(* IEC 61131-3 sources: SRCI/RobotLibrary/Library/Functions/Convert/Misc, 18 files *)

(* ---- ArmConfigParameterToBytes.st ---- *)
FUNCTION ArmConfigParameterToBytes : ARRAY[0..1] of BYTE
// -------------------------------------------------------------------------
//  SRCI Robot Library
// -------------------------------------------------------------------------
//
//  Object:      ArmConfigParameterToBytes
//  Author:      Thorsten Brach
//  Date:        2025-01-30
//
//  Description:
//
//
//  Copyright:
//    (C) 2025 Thorsten Brach. All rights reserved
//             Licensed under the LGPL-3.0 license.
//
//  Disclaimer:
//    This project is provided without any guarantee and can be used for
//    private and commercial purposes. Any use is at the user’s
//    own risk and responsibility.
//
// -------------------------------------------------------------------------
VAR_INPUT
 /// ArmConfigParameter
 Value: ArmConfigParameter;
END_VAR

  ArmConfigParameterToBytes[0].0 := Value.Shoulder.0;
  ArmConfigParameterToBytes[0].1 := Value.Shoulder.1;
  ArmConfigParameterToBytes[0].2 := Value.Shoulder.2;
  ArmConfigParameterToBytes[0].3 := Value.Shoulder.3;
  ArmConfigParameterToBytes[0].4 := Value.Elbow.0;
  ArmConfigParameterToBytes[0].5 := Value.Elbow.1;
  ArmConfigParameterToBytes[0].6 := Value.Elbow.2;
  ArmConfigParameterToBytes[0].7 := Value.Elbow.3;
  ArmConfigParameterToBytes[1].0 := Value.Wrist.0;
  ArmConfigParameterToBytes[1].1 := Value.Wrist.1;
  ArmConfigParameterToBytes[1].2 := Value.Wrist.2;
  ArmConfigParameterToBytes[1].3 := Value.Wrist.3;
  ArmConfigParameterToBytes[1].4 := FALSE;
  ArmConfigParameterToBytes[1].5 := FALSE;
  ArmConfigParameterToBytes[1].6 := FALSE;
  ArmConfigParameterToBytes[1].7 := FALSE;

END_FUNCTION

(* ---- BytesToRCSupportedFunctions.st ---- *)
FUNCTION BytesToRCSupportedFunctions : RCSupportedFunctions
// -------------------------------------------------------------------------
//  SRCI Robot Library
// -------------------------------------------------------------------------
//
//  Object:      BytesToRCSupportedFunctions
//  Author:      Thorsten Brach
//  Date:        2024-12-18
//
//  Description:
//
//
//  Copyright:
//    (C) 2024 Thorsten Brach. All rights reserved
//             Licensed under the LGPL-3.0 license.
//
//  Disclaimer:
//    This project is provided without any guarantee and can be used for
//    private and commercial purposes. Any use is at the user’s
//    own risk and responsibility.
//
// -------------------------------------------------------------------------
VAR_INPUT
  Bytes : ARRAY [0..18] OF BYTE;
END_VAR

  // Byte 00 - Bit 0
  BytesToRCSupportedFunctions.Reserved                   := Bytes[00].0;
  // Byte 00 - Bit 1
  BytesToRCSupportedFunctions.ReadRobotData              := Bytes[00].1;
  // Byte 00 - Bit 2
  BytesToRCSupportedFunctions.EnableRobot                := Bytes[00].2;
  // Byte 00 - Bit 3
  BytesToRCSupportedFunctions.GroupReset                 := Bytes[00].3;
  // Byte 00 - Bit 4
  BytesToRCSupportedFunctions.ReadActualPosition         := Bytes[00].4;
  // Byte 00 - Bit 5
  BytesToRCSupportedFunctions.ReadActualPositionCyclic   := Bytes[00].5;
  // Byte 00 - Bit 6
  BytesToRCSupportedFunctions.ExchangeConfiguration      := Bytes[00].6;
  // Byte 00 - Bit 7
  BytesToRCSupportedFunctions.SetSequence                := Bytes[00].7;

  // Byte 01 - Bit 0
  BytesToRCSupportedFunctions.ChangeSpeedOverride        := Bytes[01].0;
  // Byte 01 - Bit 1
  BytesToRCSupportedFunctions.ReadMessages               := Bytes[01].1;
  // Byte 01 - Bit 2
  BytesToRCSupportedFunctions.ReadRobotReferenceDynamics := Bytes[01].2;
  // Byte 01 - Bit 3
  BytesToRCSupportedFunctions.WriteFrameData             := Bytes[01].3;
  // Byte 01 - Bit 4
  BytesToRCSupportedFunctions.WriteToolData              := Bytes[01].4;
  // Byte 01 - Bit 5
  BytesToRCSupportedFunctions.WriteLoadData              := Bytes[01].5;
  // Byte 01 - Bit 6
  BytesToRCSupportedFunctions.WriteRobotReferenceDynamics:= Bytes[01].6;
  // Byte 01 - Bit 7
  BytesToRCSupportedFunctions.WriteRobotDefaultDynamics  := Bytes[01].7;

  // Byte 02 - Bit 0
  BytesToRCSupportedFunctions.ReadRobotDefaultDynamics   := Bytes[02].0;
  // Byte 02 - Bit 1
  BytesToRCSupportedFunctions.ReadFrameData              := Bytes[02].1;
  // Byte 02 - Bit 2
  BytesToRCSupportedFunctions.ReadToolData               := Bytes[02].2;
  // Byte 02 - Bit 3
  BytesToRCSupportedFunctions.ReadLoadData               := Bytes[02].3;
  // Byte 02 - Bit 4
  BytesToRCSupportedFunctions.ReadRobotSWLimits          := Bytes[02].4;
  // Byte 02 - Bit 5
  BytesToRCSupportedFunctions.GroupJog                   := Bytes[02].5;
  // Byte 02 - Bit 6
  BytesToRCSupportedFunctions.MoveLinearAbsolute         := Bytes[02].6;
  // Byte 02 - Bit 7
  BytesToRCSupportedFunctions.MoveDirectAbsolute         := Bytes[02].7;

  // Byte 03 - Bit 0
  BytesToRCSupportedFunctions.MoveAxesAbsolute           := Bytes[03].0;
  // Byte 03 - Bit 1
  BytesToRCSupportedFunctions.GroupStop                  := Bytes[03].1;
  // Byte 03 - Bit 2
  BytesToRCSupportedFunctions.GroupContinue              := Bytes[03].2;
  // Byte 03 - Bit 3
  BytesToRCSupportedFunctions.GroupInterrupt             := Bytes[03].3;
  // Byte 03 - Bit 4
  BytesToRCSupportedFunctions.ReturnToPrimary            := Bytes[03].4;
  // Byte 03 - Bit 5
  BytesToRCSupportedFunctions.MoveLinearAbsoluteJ        := Bytes[03].5;
  // Byte 03 - Bit 6
  BytesToRCSupportedFunctions.MoveDirectRelative         := Bytes[03].6;
  // Byte 03 - Bit 7
  BytesToRCSupportedFunctions.MoveAxesRelative           := Bytes[03].7;

  // Byte 04 - Bit 0
  BytesToRCSupportedFunctions.MoveCircularAbsolute       := Bytes[04].0;
  // Byte 04 - Bit 1
  BytesToRCSupportedFunctions.MoveCircularRelative       := Bytes[04].1;
  // Byte 04 - Bit 2
  BytesToRCSupportedFunctions.MoveLinearOffset           := Bytes[04].2;
  // Byte 04 - Bit 3
  BytesToRCSupportedFunctions.MoveDirectOffset           := Bytes[04].3;
  // Byte 04 - Bit 4
  BytesToRCSupportedFunctions.WaitTime                   := Bytes[04].4;
  // Byte 04 - Bit 5
  BytesToRCSupportedFunctions.ReadDigitalInputs          := Bytes[04].5;
  // Byte 04 - Bit 6
  BytesToRCSupportedFunctions.ReadDigitalOutputs         := Bytes[04].6;
  // Byte 04 - Bit 7
  BytesToRCSupportedFunctions.WriteDigitalOutputs        := Bytes[04].7;

  // Byte 05 - Bit 0
  BytesToRCSupportedFunctions.ReadIntegers               := Bytes[05].0;
  // Byte 05 - Bit 1
  BytesToRCSupportedFunctions.ReadReals                  := Bytes[05].1;
  // Byte 05 - Bit 2
  BytesToRCSupportedFunctions.WriteIntegers              := Bytes[05].2;
  // Byte 05 - Bit 3
  BytesToRCSupportedFunctions.WriteReals                 := Bytes[05].3;
  // Byte 05 - Bit 4
  BytesToRCSupportedFunctions.MoveLinearCam              := Bytes[05].4;
  // Byte 05 - Bit 5
  BytesToRCSupportedFunctions.MoveDirectCam              := Bytes[05].5;
  // Byte 05 - Bit 6
  BytesToRCSupportedFunctions.MoveCircularCam            := Bytes[05].6;
  // Byte 05 - Bit 7
  BytesToRCSupportedFunctions.SetTriggerRegister         := Bytes[05].7;

  // Byte 06 - Bit 0
  BytesToRCSupportedFunctions.SetTriggerLimit            := Bytes[06].0;
  // Byte 06 - Bit 1
  BytesToRCSupportedFunctions.SetTriggerUser             := Bytes[06].1;
  // Byte 06 - Bit 2
  BytesToRCSupportedFunctions.SetTriggerError            := Bytes[06].2;
  // Byte 06 - Bit 3
  BytesToRCSupportedFunctions.ReactAtTrigger             := Bytes[06].3;
  // Byte 06 - Bit 4
  BytesToRCSupportedFunctions.WaitForTrigger             := Bytes[06].4;
  // Byte 06 - Bit 5
  BytesToRCSupportedFunctions.ReadSystemVariable         := Bytes[06].5;
  // Byte 06 - Bit 6
  BytesToRCSupportedFunctions.WriteSystemVariable        := Bytes[06].6;
  // Byte 06 - Bit 7
  BytesToRCSupportedFunctions.CalculateForwardKinematic  := Bytes[06].7;

  // Byte 07 - Bit 0
  BytesToRCSupportedFunctions.CalculateInverseKinematic  := Bytes[07].0;
  // Byte 07 - Bit 1
  BytesToRCSupportedFunctions.CalculateCartesianPosition := Bytes[07].1;
  // Byte 07 - Bit 2
  BytesToRCSupportedFunctions.CalculateTool              := Bytes[07].2;
  // Byte 07 - Bit 3
  BytesToRCSupportedFunctions.CalculateFrame             := Bytes[07].3;
  // Byte 07 - Bit 4
  BytesToRCSupportedFunctions.ActivateNextCommand        := Bytes[07].4;
  // Byte 07 - Bit 5
  BytesToRCSupportedFunctions.ShiftPosition              := Bytes[07].5;
  // Byte 07 - Bit 6
  BytesToRCSupportedFunctions.CallSubprogram             := Bytes[07].6;
  // Byte 07 - Bit 7
  BytesToRCSupportedFunctions.MoveLinearRelative         := Bytes[07].7;

  // Byte 08 - Bit 0
  BytesToRCSupportedFunctions.WriteCallSubprogramCyclic  := Bytes[08].0;
  // Byte 08 - Bit 1
  BytesToRCSupportedFunctions.ReadCallSubprogramCyclic   := Bytes[08].1;
  // Byte 08 - Bit 2
  BytesToRCSupportedFunctions.StopSubprogram             := Bytes[08].2;
  // Byte 08 - Bit 3
  BytesToRCSupportedFunctions.ReadDHParameter            := Bytes[08].3;
  // Byte 08 - Bit 4
  BytesToRCSupportedFunctions.RestartController          := Bytes[08].4;
  // Byte 08 - Bit 5
  BytesToRCSupportedFunctions.ReadActualTCPVelocity      := Bytes[08].5;
  // Byte 08 - Bit 6
  BytesToRCSupportedFunctions.UserLogin                  := Bytes[08].6;
  // Byte 08 - Bit 7
  BytesToRCSupportedFunctions.SwitchLanguage             := Bytes[08].7;

  // Byte 09 - Bit 0
  BytesToRCSupportedFunctions.WriteRobotSWLimits         := Bytes[09].0;
  // Byte 09 - Bit 1
  BytesToRCSupportedFunctions.SetOperationMode           := Bytes[09].1;
  // Byte 09 - Bit 2
  BytesToRCSupportedFunctions.ReadWorkArea               := Bytes[09].2;
  // Byte 09 - Bit 3
  BytesToRCSupportedFunctions.WriteWorkArea              := Bytes[09].3;
  // Byte 09 - Bit 4
  BytesToRCSupportedFunctions.ActivateWorkArea           := Bytes[09].4;
  // Byte 09 - Bit 5
  BytesToRCSupportedFunctions.MonitorWorkArea            := Bytes[09].5;
  // Byte 09 - Bit 6
  BytesToRCSupportedFunctions.MoveApproachLinear         := Bytes[09].6;
  // Byte 09 - Bit 7
  BytesToRCSupportedFunctions.MoveDepartLinear           := Bytes[09].7;

  // Byte 10 - Bit 0
  BytesToRCSupportedFunctions.MoveApproachDirect         := Bytes[10].0;
  // Byte 10 - Bit 1
  BytesToRCSupportedFunctions.MoveDepartDirect           := Bytes[10].1;
  // Byte 10 - Bit 2
  BytesToRCSupportedFunctions.SearchHardstop             := Bytes[10].2;
  // Byte 10 - Bit 3
  BytesToRCSupportedFunctions.SearchHardstopJ            := Bytes[10].3;
  // Byte 10 - Bit 4
  BytesToRCSupportedFunctions.MovePickPlaceLinear        := Bytes[10].4;
  // Byte 10 - Bit 5
  BytesToRCSupportedFunctions.MovePickPlaceDirect        := Bytes[10].5;
  // Byte 10 - Bit 6
  BytesToRCSupportedFunctions.ActivateConveyorTracking   := Bytes[10].6;
  // Byte 10 - Bit 7
  BytesToRCSupportedFunctions.RedefineTrackingPosition   := Bytes[10].7;

  // Byte 11 - Bit 0
  BytesToRCSupportedFunctions.SyncToConveyor             := Bytes[11].0;
  // Byte 11 - Bit 1
  BytesToRCSupportedFunctions.ConfigureConveyor          := Bytes[11].1;
  // Byte 11 - Bit 2
  BytesToRCSupportedFunctions.MoveSuperImposed           := Bytes[11].2;
  // Byte 11 - Bit 3
  BytesToRCSupportedFunctions.MoveSuperImposedDynamic    := Bytes[11].3;
  // Byte 11 - Bit 4
  BytesToRCSupportedFunctions.ReadAnalogInput            := Bytes[11].4;
  // Byte 11 - Bit 5
  BytesToRCSupportedFunctions.ReadAnalogOutput           := Bytes[11].5;
  // Byte 11 - Bit 6
  BytesToRCSupportedFunctions.WriteAnalogOutput          := Bytes[11].6;
  // Byte 11 - Bit 7
  BytesToRCSupportedFunctions.MeasuringInput             := Bytes[11].7;

  // Byte 12 - Bit 0
  BytesToRCSupportedFunctions.AbortMeasuringInput        := Bytes[12].0;
  // Byte 12 - Bit 1
  BytesToRCSupportedFunctions.SetTriggerMotion           := Bytes[12].1;
  // Byte 12 - Bit 2
  BytesToRCSupportedFunctions.OpenBrake                  := Bytes[12].2;
  // Byte 12 - Bit 3
  BytesToRCSupportedFunctions.PathAccuracyMode           := Bytes[12].3;
  // Byte 12 - Bit 4
  BytesToRCSupportedFunctions.AvoidSingularity           := Bytes[12].4;
  // Byte 12 - Bit 5
  BytesToRCSupportedFunctions.ForceControl               := Bytes[12].5;
  // Byte 12 - Bit 6
  BytesToRCSupportedFunctions.ForceLimit                 := Bytes[12].6;
  // Byte 12 - Bit 7
  BytesToRCSupportedFunctions.ReadActualForce            := Bytes[12].7;

  // Byte 13 - Bit 0
  BytesToRCSupportedFunctions.BrakeTest                  := Bytes[13].0;
  // Byte 13 - Bit 1
  BytesToRCSupportedFunctions.SoftSwitchTCP              := Bytes[13].1;
  // Byte 13 - Bit 2
  BytesToRCSupportedFunctions.CreateSpline               := Bytes[13].2;
  // Byte 13 - Bit 3
  BytesToRCSupportedFunctions.DeleteSpline               := Bytes[13].3;
  // Byte 13 - Bit 4
  BytesToRCSupportedFunctions.MoveSpline                 := Bytes[13].4;
  // Byte 13 - Bit 5
  BytesToRCSupportedFunctions.DynamicSpline              := Bytes[13].5;
  // Byte 13 - Bit 6
  BytesToRCSupportedFunctions.LoadMeasurementAutomatic   := Bytes[13].6;
  // Byte 13 - Bit 7
  BytesToRCSupportedFunctions.LoadMeasurementSequential  := Bytes[13].7;

  // Byte 14 - Bit 0
  BytesToRCSupportedFunctions.CollisionDetection         := Bytes[14].0;
  // Byte 14 - Bit 1
  BytesToRCSupportedFunctions.FreeDrive                  := Bytes[14].1;
  // Byte 14 - Bit 2
  BytesToRCSupportedFunctions.UnitMeasurement            := Bytes[14].2;
  // Byte 14 - Bit 3
  BytesToRCSupportedFunctions.Byte14Bit03                := Bytes[14].3;
  // Byte 14 - Bit 4
  BytesToRCSupportedFunctions.Byte14Bit04                := Bytes[14].4;
  // Byte 14 - Bit 5
  BytesToRCSupportedFunctions.Byte14Bit05                := Bytes[14].5;
  // Byte 14 - Bit 6
  BytesToRCSupportedFunctions.Byte14Bit06                := Bytes[14].6;
  // Byte 14 - Bit 7
  BytesToRCSupportedFunctions.Byte14Bit07                := Bytes[14].7;

  // Byte 15 - Bit 0
  BytesToRCSupportedFunctions.Byte15Bit00                := Bytes[15].0;
  // Byte 15 - Bit 1
  BytesToRCSupportedFunctions.Byte15Bit01                := Bytes[15].1;
  // Byte 15 - Bit 2
  BytesToRCSupportedFunctions.Byte15Bit02                := Bytes[15].2;
  // Byte 15 - Bit 3
  BytesToRCSupportedFunctions.Byte15Bit03                := Bytes[15].3;
  // Byte 15 - Bit 4
  BytesToRCSupportedFunctions.Byte15Bit04                := Bytes[15].4;
  // Byte 15 - Bit 5
  BytesToRCSupportedFunctions.Byte15Bit05                := Bytes[15].5;
  // Byte 15 - Bit 6
  BytesToRCSupportedFunctions.Byte15Bit06                := Bytes[15].6;
  // Byte 15 - Bit 7
  BytesToRCSupportedFunctions.Byte15Bit07                := Bytes[15].7;

  // Byte 16 - Bit 0
  BytesToRCSupportedFunctions.Byte16Bit00                := Bytes[16].0;
  // Byte 15 - Bit 1
  BytesToRCSupportedFunctions.Byte16Bit01                := Bytes[16].1;
  // Byte 15 - Bit 2
  BytesToRCSupportedFunctions.Byte16Bit02                := Bytes[16].2;
  // Byte 15 - Bit 3
  BytesToRCSupportedFunctions.Byte16Bit03                := Bytes[16].3;
  // Byte 15 - Bit 4
  BytesToRCSupportedFunctions.Byte16Bit04                := Bytes[16].4;
  // Byte 15 - Bit 5
  BytesToRCSupportedFunctions.Byte16Bit05                := Bytes[16].5;
  // Byte 15 - Bit 6
  BytesToRCSupportedFunctions.Byte16Bit06                := Bytes[16].6;
  // Byte 15 - Bit 7
  BytesToRCSupportedFunctions.Byte16Bit07                := Bytes[16].7;

  // Byte 17 - Bit 0
  BytesToRCSupportedFunctions.Byte17Bit00                := Bytes[17].0;
  // Byte 17 - Bit 1
  BytesToRCSupportedFunctions.Byte17Bit01                := Bytes[17].1;
  // Byte 17 - Bit 2
  BytesToRCSupportedFunctions.Byte17Bit02                := Bytes[17].2;
  // Byte 17 - Bit 3
  BytesToRCSupportedFunctions.Byte17Bit03                := Bytes[17].3;
  // Byte 17 - Bit 4
  BytesToRCSupportedFunctions.Byte17Bit04                := Bytes[17].4;
  // Byte 17 - Bit 5
  BytesToRCSupportedFunctions.Byte17Bit05                := Bytes[17].5;
  // Byte 17 - Bit 6
  BytesToRCSupportedFunctions.Byte17Bit06                := Bytes[17].6;
  // Byte 17 - Bit 7
  BytesToRCSupportedFunctions.Byte17Bit07                := Bytes[17].7;

  // Byte 18 - Bit 0
  BytesToRCSupportedFunctions.Byte18Bit00                := Bytes[18].0;
  // Byte 18 - Bit 1
  BytesToRCSupportedFunctions.Byte18Bit01                := Bytes[18].1;
  // Byte 18 - Bit 2
  BytesToRCSupportedFunctions.Byte18Bit02                := Bytes[18].2;
  // Byte 18 - Bit 3
  BytesToRCSupportedFunctions.Byte18Bit03                := Bytes[18].3;
  // Byte 18 - Bit 4
  BytesToRCSupportedFunctions.Byte18Bit04                := Bytes[18].4;
  // Byte 18 - Bit 5
  BytesToRCSupportedFunctions.Byte18Bit05                := Bytes[18].5;
  // Byte 18 - Bit 6
  BytesToRCSupportedFunctions.Byte18Bit06                := Bytes[18].6;
  // Byte 18 - Bit 7
  BytesToRCSupportedFunctions.Byte18Bit07                := Bytes[18].7;

END_FUNCTION

(* ---- ByteToAxisExternalUnit.st ---- *)
FUNCTION ByteToAxisExternalUnit : AxisExternalUnit
// -------------------------------------------------------------------------
//  SRCI Robot Library
// -------------------------------------------------------------------------
//
//  Object:      ByteToAxisExternalUnit
//  Author:      Thorsten Brach
//  Date:        2025-03-23
//
//  Description:
//
//
//  Copyright:
//    (C) 2025 Thorsten Brach. All rights reserved
//             Licensed under the LGPL-3.0 license.
//
//  Disclaimer:
//    This project is provided without any guarantee and can be used for
//    private and commercial purposes. Any use is at the user’s
//    own risk and responsibility.
//
// -------------------------------------------------------------------------
VAR_INPUT
  AxisExternalUnit : BYTE;
END_VAR

  ByteToAxisExternalUnit.E1.0 := AxisExternalUnit.1;
  ByteToAxisExternalUnit.E2.0 := AxisExternalUnit.2;
  ByteToAxisExternalUnit.E3.0 := AxisExternalUnit.3;
  ByteToAxisExternalUnit.E4.0 := AxisExternalUnit.4;
  ByteToAxisExternalUnit.E5.0 := AxisExternalUnit.5;
  ByteToAxisExternalUnit.E6.0 := AxisExternalUnit.6;

END_FUNCTION

(* ---- ByteToAxisExternalUsed.st ---- *)
FUNCTION ByteToAxisExternalUsed : AxisExternalUsed
// -------------------------------------------------------------------------
//  SRCI Robot Library
// -------------------------------------------------------------------------
//
//  Object:      ByteToAxisExternalUsed
//  Author:      Thorsten Brach
//  Date:        2025-03-23
//
//  Description:
//
//
//  Copyright:
//    (C) 2025 Thorsten Brach. All rights reserved
//             Licensed under the LGPL-3.0 license.
//
//  Disclaimer:
//    This project is provided without any guarantee and can be used for
//    private and commercial purposes. Any use is at the user’s
//    own risk and responsibility.
//
// -------------------------------------------------------------------------
VAR_INPUT
  AxisExternalUsed : BYTE;
END_VAR

  ByteToAxisExternalUsed.E1 := AxisExternalUsed.1;
  ByteToAxisExternalUsed.E2 := AxisExternalUsed.2;
  ByteToAxisExternalUsed.E3 := AxisExternalUsed.3;
  ByteToAxisExternalUsed.E4 := AxisExternalUsed.4;
  ByteToAxisExternalUsed.E5 := AxisExternalUsed.5;
  ByteToAxisExternalUsed.E6 := AxisExternalUsed.6;

END_FUNCTION

(* ---- ByteToAxisJointUnit.st ---- *)
FUNCTION ByteToAxisJointUnit : AxisJointUnit
// -------------------------------------------------------------------------
//  SRCI Robot Library
// -------------------------------------------------------------------------
//
//  Object:      ByteToAxisJointUnit
//  Author:      Thorsten Brach
//  Date:        2025-03-23
//
//  Description:
//
//
//  Copyright:
//    (C) 2025 Thorsten Brach. All rights reserved
//             Licensed under the LGPL-3.0 license.
//
//  Disclaimer:
//    This project is provided without any guarantee and can be used for
//    private and commercial purposes. Any use is at the user’s
//    own risk and responsibility.
//
// -------------------------------------------------------------------------
VAR_INPUT
  AxisJointUnit : BYTE;
END_VAR

  ByteToAxisJointUnit.J2.0 := AxisJointUnit.1;
  ByteToAxisJointUnit.J2.0 := AxisJointUnit.2;
  ByteToAxisJointUnit.J3.0 := AxisJointUnit.3;
  ByteToAxisJointUnit.J4.0 := AxisJointUnit.4;
  ByteToAxisJointUnit.J5.0 := AxisJointUnit.5;
  ByteToAxisJointUnit.J6.0 := AxisJointUnit.6;

END_FUNCTION

(* ---- ByteToAxisJointUsed.st ---- *)
FUNCTION ByteToAxisJointUsed : AxisJointUsed
// -------------------------------------------------------------------------
//  SRCI Robot Library
// -------------------------------------------------------------------------
//
//  Object:      ByteToAxisJointUsed
//  Author:      Thorsten Brach
//  Date:        2025-03-23
//
//  Description:
//
//
//  Copyright:
//    (C) 2025 Thorsten Brach. All rights reserved
//             Licensed under the LGPL-3.0 license.
//
//  Disclaimer:
//    This project is provided without any guarantee and can be used for
//    private and commercial purposes. Any use is at the user’s
//    own risk and responsibility.
//
// -------------------------------------------------------------------------
VAR_INPUT
  AxisJointUsed : BYTE;
END_VAR

  ByteToAxisJointUsed.J1 := AxisJointUsed.1;
  ByteToAxisJointUsed.J2 := AxisJointUsed.2;
  ByteToAxisJointUsed.J3 := AxisJointUsed.3;
  ByteToAxisJointUsed.J4 := AxisJointUsed.4;
  ByteToAxisJointUsed.J5 := AxisJointUsed.5;
  ByteToAxisJointUsed.J6 := AxisJointUsed.6;

END_FUNCTION

(* ---- CombineBytesToUint.st ---- *)
FUNCTION CombineBytesToUint : UINT
// -------------------------------------------------------------------------
//  SRCI Robot Library
// -------------------------------------------------------------------------
//
//  Object:      CombineBytes
//  Author:      Thorsten Brach
//  Date:        2024-09-03
//
//  Description:
//
//
//  Copyright:
//    (C) 2024 Thorsten Brach. All rights reserved
//             Licensed under the LGPL-3.0 license.
//
//  Disclaimer:
//    This project is provided without any guarantee and can be used for
//    private and commercial purposes. Any use is at the user’s
//    own risk and responsibility.
//
// -------------------------------------------------------------------------
VAR_INPUT
  /// Byte to add as high byte
  HiByte : BYTE;
  /// Byte to add as low byte
  LoByte : BYTE;
END_VAR

  CombineBytesToUint.0  := LoByte.0;
  CombineBytesToUint.1  := LoByte.1;
  CombineBytesToUint.2  := LoByte.2;
  CombineBytesToUint.3  := LoByte.3;
  CombineBytesToUint.4  := LoByte.4;
  CombineBytesToUint.5  := LoByte.5;
  CombineBytesToUint.6  := LoByte.6;
  CombineBytesToUint.7  := LoByte.7;

  CombineBytesToUint.8  := HiByte.0;
  CombineBytesToUint.9  := HiByte.1;
  CombineBytesToUint.10 := HiByte.2;
  CombineBytesToUint.11 := HiByte.3;
  CombineBytesToUint.12 := HiByte.4;
  CombineBytesToUint.13 := HiByte.5;
  CombineBytesToUint.14 := HiByte.6;
  CombineBytesToUint.15 := HiByte.7;

END_FUNCTION

(* ---- CombineHalfSints.st ---- *)
FUNCTION CombineHalfSints : USINT
// -------------------------------------------------------------------------
//  SRCI Robot Library
// -------------------------------------------------------------------------
//
//  Object:      CombineHalfSints
//  Author:      Thorsten Brach
//  Date:        2025-02-02
//
//  Description:
//
//
//  Copyright:
//    (C) 2025 Thorsten Brach. All rights reserved
//             Licensed under the LGPL-3.0 license.
//
//  Disclaimer:
//    This project is provided without any guarantee and can be used for
//    private and commercial purposes. Any use is at the user’s
//    own risk and responsibility.
//
// -------------------------------------------------------------------------
VAR_INPUT
  /// Half-Sint to add to the upper 4 Bit
  HalfSintHi : SINT;
  /// Half-Sint to add to the lower 4 Bit
  HalfSintLo : SINT;
END_VAR

  // merage ParSeq and Priority to combined variable
  CombineHalfSints.0 := HalfSintLo.0;
  CombineHalfSints.1 := HalfSintLo.1;
  CombineHalfSints.2 := HalfSintLo.2;
  CombineHalfSints.3 := HalfSintLo.3;

  CombineHalfSints.4 := HalfSintHi.0;
  CombineHalfSints.5 := HalfSintHi.1;
  CombineHalfSints.6 := HalfSintHi.2;
  CombineHalfSints.7 := HalfSintHi.3;

END_FUNCTION

(* ---- DwordToRaStatusWord.st ---- *)
FUNCTION DwordToRaStatusWord : RaStatusWord
// -------------------------------------------------------------------------
//  SRCI Robot Library
// -------------------------------------------------------------------------
//
//  Object:      DwordToRaStatusWord
//  Author:      Thorsten Brach
//  Date:        2024-11-16
//
//  Description:
//
//
//  Copyright:
//    (C) 2024 Thorsten Brach. All rights reserved
//             Licensed under the LGPL-3.0 license.
//
//  Disclaimer:
//    This project is provided without any guarantee and can be used for
//    private and commercial purposes. Any use is at the user’s
//    own risk and responsibility.
//
// -------------------------------------------------------------------------
VAR_INPUT
  /// Value
  Value : DWORD;
END_VAR

  DwordToRaStatusWord.IsMoving                 := Value.00;
  DwordToRaStatusWord.PrimarySequencePaused    := Value.01;
  DwordToRaStatusWord.InPrimaryPos             := Value.02;
  DwordToRaStatusWord.SecondarySequenceActive  := Value.03;
  DwordToRaStatusWord.IsBlending               := Value.04;
  DwordToRaStatusWord.ErrorPending             := Value.05;
  DwordToRaStatusWord.RestartInProgress        := Value.06;
  DwordToRaStatusWord.Enabled                  := Value.07;
  DwordToRaStatusWord.RaSequenceState.0        := Value.08;
  DwordToRaStatusWord.RaSequenceState.1        := Value.09;
  DwordToRaStatusWord.OperationMode.0          := Value.10;
  DwordToRaStatusWord.OperationMode.1          := Value.11;
  DwordToRaStatusWord.OperationMode.2          := Value.12;
  DwordToRaStatusWord.CollisionDetectedEnabled := Value.13;
  DwordToRaStatusWord.CollisionDetected        := Value.14;
  DwordToRaStatusWord.RestartRequested         := Value.15;
  DwordToRaStatusWord.Accelerating             := Value.16;
  DwordToRaStatusWord.Decelerating             := Value.17;
  DwordToRaStatusWord.ConstantVelocity         := Value.18;
  DwordToRaStatusWord.Bit19                    := Value.19;
  DwordToRaStatusWord.Bit20                    := Value.20;
  DwordToRaStatusWord.Bit21                    := Value.21;
  DwordToRaStatusWord.Bit22                    := Value.22;
  DwordToRaStatusWord.Bit23                    := Value.23;
  DwordToRaStatusWord.Bit24                    := Value.24;
  DwordToRaStatusWord.Bit25                    := Value.25;
  DwordToRaStatusWord.Bit26                    := Value.26;
  DwordToRaStatusWord.Bit27                    := Value.27;
  DwordToRaStatusWord.Bit28                    := Value.28;
  DwordToRaStatusWord.Bit29                    := Value.29;
  DwordToRaStatusWord.Bit30                    := Value.30;
  DwordToRaStatusWord.Bit31                    := Value.31;

END_FUNCTION

(* ---- PERCENT_INT_TO_REAL.st ---- *)
FUNCTION PERCENT_INT_TO_REAL : REAL
// -------------------------------------------------------------------------
//  SRCI Robot Library
// -------------------------------------------------------------------------
//
//  Object:      PERCENT_INT_TO_REAL
//  Author:      Thorsten Brach
//  Date:        2025-02-07
//
//  Description:
//
//
//  Copyright:
//    (C) 2025 Thorsten Brach. All rights reserved
//             Licensed under the LGPL-3.0 license.
//
//  Disclaimer:
//    This project is provided without any guarantee and can be used for
//    private and commercial purposes. Any use is at the user’s
//    own risk and responsibility.
//
// -------------------------------------------------------------------------
VAR_INPUT
  /// Percent value to convert
  Value    : INT;
  /// value is an optional parameter ?
  IsOptional : BOOL;
END_VAR

  IF ( Value = 16#FFFF ) AND (IsOptional)// 16#FFFF for not supported values
  THEN
    PERCENT_INT_TO_REAL := -1.0;
    RETURN;
  END_IF

  PERCENT_INT_TO_REAL := INT_TO_REAL(Value) / RobotLibraryConstants.REAL_CONVERSION_FACTOR; {warning 'ToDo: check conversation is correct ?'}

END_FUNCTION

(* ---- PERCENT_UINT_TO_REAL.st ---- *)
FUNCTION PERCENT_UINT_TO_REAL : REAL
// -------------------------------------------------------------------------
//  SRCI Robot Library
// -------------------------------------------------------------------------
//
//  Object:      PERCENT_UINT_TO_REAL
//  Author:      Thorsten Brach
//  Date:        2025-04-02
//
//  Description:
//
//
//  Copyright:
//    (C) 2025 Thorsten Brach. All rights reserved
//             Licensed under the LGPL-3.0 license.
//
//  Disclaimer:
//    This project is provided without any guarantee and can be used for
//    private and commercial purposes. Any use is at the user’s
//    own risk and responsibility.
//
// -------------------------------------------------------------------------
VAR_INPUT
  /// Percent value to convert
  Value    : UINT;
  /// value is an optional parameter ?
  IsOptional : BOOL;
END_VAR

  IF (( Value = 16#FFFF_FFFF ) AND (IsOptional)) OR // 16#FFFF_FFFF for not supported values
     (( Value = 16#0000_FFFF ) AND (IsOptional))    // 16#0000_FFFF for not supported values
  THEN
    PERCENT_UINT_TO_REAL := -1.0;
    RETURN;
  END_IF

  PERCENT_UINT_TO_REAL := UINT_TO_REAL(Value) / RobotLibraryConstants.REAL_CONVERSION_FACTOR;

END_FUNCTION

(* ---- REAL_TO_PERCENT_INT.st ---- *)
FUNCTION REAL_TO_PERCENT_INT : INT
// -------------------------------------------------------------------------
//  SRCI Robot Library
// -------------------------------------------------------------------------
//
//  Object:      REAL_TO_PERCENT_INT
//  Author:      Thorsten Brach
//  Date:        2025-02-07
//
//  Description:
//
//
//  Copyright:
//    (C) 2025 Thorsten Brach. All rights reserved
//             Licensed under the LGPL-3.0 license.
//
//  Disclaimer:
//    This project is provided without any guarantee and can be used for
//    private and commercial purposes. Any use is at the user’s
//    own risk and responsibility.
//
// -------------------------------------------------------------------------
VAR_INPUT
  /// Percent value to convert
  Value      : REAL;
  /// value is an optional parameter ?
  IsOptional : BOOL;
END_VAR

  IF ( Value = -1.0)  AND (IsOptional)// 16#FFFF for not supported values
  THEN
    REAL_TO_PERCENT_INT := UINT_TO_INT(16#FFFF);
    RETURN;
  END_IF

  REAL_TO_PERCENT_INT := REAL_TO_INT(Value * RobotLibraryConstants.REAL_CONVERSION_FACTOR);

END_FUNCTION

(* ---- REAL_TO_PERCENT_UINT.st ---- *)
FUNCTION REAL_TO_PERCENT_UINT : UINT
// -------------------------------------------------------------------------
//  SRCI Robot Library
// -------------------------------------------------------------------------
//
//  Object:      REAL_TO_PERCENT_UINT
//  Author:      Thorsten Brach
//  Date:        2025-02-07
//
//  Description:
//
//
//  Copyright:
//    (C) 2025 Thorsten Brach. All rights reserved
//             Licensed under the LGPL-3.0 license.
//
//  Disclaimer:
//    This project is provided without any guarantee and can be used for
//    private and commercial purposes. Any use is at the user’s
//    own risk and responsibility.
//
// -------------------------------------------------------------------------
VAR_INPUT
  /// Percent value to convert
  Value      : REAL;
  /// value is an optional parameter ?
  IsOptional : BOOL;
END_VAR

  IF ( Value = -1.0)  AND (IsOptional)// 16#FFFF for not supported values
  THEN
    REAL_TO_PERCENT_UINT := 16#FFFF;
    RETURN;
  END_IF

  REAL_TO_PERCENT_UINT := REAL_TO_UINT(Value * RobotLibraryConstants.REAL_CONVERSION_FACTOR);

END_FUNCTION

(* ---- SyncModesToDataEnableSync.st ---- *)
FUNCTION SyncModesToDataEnableSync : DataEnableSync
// -------------------------------------------------------------------------
//  SRCI Robot Library
// -------------------------------------------------------------------------
//
//  Object:      SyncModesToDataEnableSync
//  Author:      Thorsten Brach
//  Date:        2025-04-22
//
//  Description:
//
//
//  Copyright:
//    (C) 2025 Thorsten Brach. All rights reserved
//             Licensed under the LGPL-3.0 license.
//
//  Disclaimer:
//    This project is provided without any guarantee and can be used for
//    private and commercial purposes. Any use is at the user’s
//    own risk and responsibility.
//
// -------------------------------------------------------------------------
VAR_INPUT
  /// Synchronization Modes
  Value : SynchronizationModes;
END_VAR

  SyncModesToDataEnableSync.EnableSyncTool              := Value.Tool             [SyncTime.DURING_START_UP] > SyncMode.NO_SYNCHRONIZATION OR
                                                           Value.Tool             [SyncTime. AFTER_START_UP] > SyncMode.NO_SYNCHRONIZATION;
  SyncModesToDataEnableSync.EnableSyncFrame             := Value.Frame            [SyncTime.DURING_START_UP] > SyncMode.NO_SYNCHRONIZATION OR
                                                           Value.Frame            [SyncTime. AFTER_START_UP] > SyncMode.NO_SYNCHRONIZATION;
  SyncModesToDataEnableSync.EnableSyncLoad              := Value.Load             [SyncTime.DURING_START_UP] > SyncMode.NO_SYNCHRONIZATION OR
                                                           Value.Load             [SyncTime. AFTER_START_UP] > SyncMode.NO_SYNCHRONIZATION;
  SyncModesToDataEnableSync.EnableSyncWorkArea          := Value.WorkAreas        [SyncTime.DURING_START_UP] > SyncMode.NO_SYNCHRONIZATION OR
                                                           Value.WorkAreas        [SyncTime. AFTER_START_UP] > SyncMode.NO_SYNCHRONIZATION;
  SyncModesToDataEnableSync.EnableSyncSWLimits          := Value.SWLimits         [SyncTime.DURING_START_UP] > SyncMode.NO_SYNCHRONIZATION OR
                                                           Value.SWLimits         [SyncTime. AFTER_START_UP] > SyncMode.NO_SYNCHRONIZATION;
  SyncModesToDataEnableSync.EnableSyncDefaultDynamics   := Value.DefaultDynamics  [SyncTime.DURING_START_UP] > SyncMode.NO_SYNCHRONIZATION OR
                                                           Value.DefaultDynamics  [SyncTime. AFTER_START_UP] > SyncMode.NO_SYNCHRONIZATION;
  SyncModesToDataEnableSync.EnableSyncReferenceDynamics := Value.ReferenceDynamics[SyncTime.DURING_START_UP] > SyncMode.NO_SYNCHRONIZATION OR
                                                           Value.ReferenceDynamics[SyncTime. AFTER_START_UP] > SyncMode.NO_SYNCHRONIZATION;

END_FUNCTION

(* ---- VersionToByte.st ---- *)
FUNCTION VersionToByte : BYTE
// -------------------------------------------------------------------------
//  SRCI Robot Library
// -------------------------------------------------------------------------
//
//  Object:      VersionToByte
//  Author:      Thorsten Brach
//  Date:        2024-06-01
//
//  Description:
//
//
//  Copyright:
//    (C) 2024 Thorsten Brach. All rights reserved
//             Licensed under the LGPL-3.0 license.
//
//  Disclaimer:
//    This project is provided without any guarantee and can be used for
//    private and commercial purposes. Any use is at the user’s
//    own risk and responsibility.
//
// -------------------------------------------------------------------------
VAR_INPUT
  /// Version
  Value : VersionStruct;
END_VAR

VAR
  _tmpByte : BYTE;
END_VAR

  // Minor version  • Features
  //                • 0..31 minor versions
  VersionToByte.0 := Value.MinorVersion.0;
  VersionToByte.1 := Value.MinorVersion.1;
  VersionToByte.2 := Value.MinorVersion.2;
  VersionToByte.3 := Value.MinorVersion.3;
  VersionToByte.4 := Value.MinorVersion.4;

  // Major version  • Breaking change
  //                • 0..7 major versions
  VersionToByte.5 := Value.MajorVersion.0;
  VersionToByte.6 := Value.MajorVersion.1;
  VersionToByte.7 := Value.MajorVersion.2;

END_FUNCTION

(* ---- WordToArmConfigElbow.st ---- *)
FUNCTION WordToArmConfigElbow : ArmConfigElbow
// -------------------------------------------------------------------------
//  SRCI Robot Library
// -------------------------------------------------------------------------
//
//  Object:      WordToArmConfigElbow
//  Author:      Thorsten Brach
//  Date:        2024-12-24
//
//  Description:
//
//
//  Copyright:
//    (C) 2024 Thorsten Brach. All rights reserved
//             Licensed under the LGPL-3.0 license.
//
//  Disclaimer:
//    This project is provided without any guarantee and can be used for
//    private and commercial purposes. Any use is at the user’s
//    own risk and responsibility.
//
// -------------------------------------------------------------------------
VAR_INPUT
  /// Value
  Value : WORD;
END_VAR

VAR
  _tmpByte : BYTE;
END_VAR

  IF ( RobotLibraryParameter.SWAP_BYTE_ORDER)
  THEN
    Value := SwapWord(Value);
  END_IF

  IF (Value.1)
  THEN
    WordToArmConfigElbow := ArmConfigElbow.DOWN;
  ELSE
    WordToArmConfigElbow := ArmConfigElbow.UP;
  END_IF

END_FUNCTION

(* ---- WordToArmConfigShoulder.st ---- *)
FUNCTION WordToArmConfigShoulder : ArmConfigShoulder
// -------------------------------------------------------------------------
//  SRCI Robot Library
// -------------------------------------------------------------------------
//
//  Object:      WordToArmConfigShoulder
//  Author:      Thorsten Brach
//  Date:        2024-12-24
//
//  Description:
//
//
//  Copyright:
//    (C) 2024 Thorsten Brach. All rights reserved
//             Licensed under the LGPL-3.0 license.
//
//  Disclaimer:
//    This project is provided without any guarantee and can be used for
//    private and commercial purposes. Any use is at the user’s
//    own risk and responsibility.
//
// -------------------------------------------------------------------------
VAR_INPUT
  /// Value
  Value : WORD;
END_VAR

VAR
  _tmpByte : BYTE;
END_VAR

  IF ( RobotLibraryParameter.SWAP_BYTE_ORDER)
  THEN
    Value := SwapWord(Value);
  END_IF

  IF (Value.0)
  THEN
    WordToArmConfigShoulder := ArmConfigShoulder.BACK;
  ELSE
    WordToArmConfigShoulder := ArmConfigShoulder.FRONT;
  END_IF

END_FUNCTION

(* ---- WordToArmConfigWrist.st ---- *)
FUNCTION WordToArmConfigWrist : ArmConfigWrist
// -------------------------------------------------------------------------
//  SRCI Robot Library
// -------------------------------------------------------------------------
//
//  Object:      WordToArmConfigWrist
//  Author:      Thorsten Brach
//  Date:        2024-12-24
//
//  Description:
//
//
//  Copyright:
//    (C) 2024 Thorsten Brach. All rights reserved
//             Licensed under the LGPL-3.0 license.
//
//  Disclaimer:
//    This project is provided without any guarantee and can be used for
//    private and commercial purposes. Any use is at the user’s
//    own risk and responsibility.
//
// -------------------------------------------------------------------------
VAR_INPUT
  /// Value
  Value : WORD;
END_VAR

VAR
  _tmpByte : BYTE;
END_VAR

  IF ( RobotLibraryParameter.SWAP_BYTE_ORDER)
  THEN
    Value := SwapWord(Value);
  END_IF

  IF (Value.2)
  THEN
    WordToArmConfigWrist := ArmConfigWrist.FLIP;
  ELSE
    WordToArmConfigWrist := ArmConfigWrist.NON_FLIP;
  END_IF

END_FUNCTION
